(* CoDeSys 2.3 export: FSETK15PUMP.EXP *)

(* POU K15/fSetK15Pump, ST *)
FUNCTION fSetK15Pump : BOOL
VAR_INPUT
	State : BOOL;
	PumpID : USINT;
END_VAR
VAR
END_VAR
	PLC160DO.K15Pump[PumpID] := State;
	(*Включить/Выключить реле насоса*)
END_FUNCTION
